INTERFACE ITFLoggingProvider

/// Add log method
{attribute 'object_name' := 'AddLog'}
METHOD AddLog : BOOL
VAR_INPUT
	/// log message 
	sText: T_MaxString;
	/// log source
	sSource: STRING;
	///	level: eLogLevelNone, eLogLevelError, eLogLevelWarning, eLogLevelInformation	
	eLevel: E_LogLevel;
END_VAR
END_METHOD

{attribute 'object_name' := 'Run'}
METHOD Run
END_METHOD

END_INTERFACE

(* stored: Version 1.1.0.1
   Itf ITFLoggingProvider: Id {d243c429-a89c-47b6-9f05-cc3d571a859b}
   Method AddLog: Id {38f0b6ec-65a4-4189-9644-75514e750fde}
   Method Run: Id {2e2fa1d8-9f8f-4441-afb9-d1d885893511} *)
